TYPE ST_HW_InOutputsSTI_EtherCAT_Conveyor :
(**************************************************************************************
 * 	Application		:	BoxControl Framework
 *	Revision		:	$Revision: 355211 $
 *	Revision date	:	$Date: 2015-09-22 11:14:21 +0200 (Tue, 22 Sep 2015) $
 *	Last changed by	:	$Author: b7bolm $
 *	URL				:	$URL: http://almscdc.swisslog.com/repo/SWPD/Development/BoxControlFramework/20_Release/trunk/01_Software/BoxControlFramework/BoxControlFramework/JumpStart/11_Library/10_Application/11_Communication/12_MFCS/11_SIS/10_Base/FB_SIS_BaseDriver.TcPOU $
 *
 *	Purpose			:	Data for conveyor Subsystem interface over EtherCAT
 *
 * ------------------------------------------------------------------------------------
 *	Copyright Swisslog [IP AG], Switzerland. All rights reserved.
 * 
 * ------------------------------------------------------------------------------------
 *	
 * 	Revision History: 
 *
 * 	VERSION			DATE			INITIALS			DESCRIPTION
 *	0.1				01.01.2001		swl					Example
 *
 **************************************************************************************)
STRUCT
	Watchdog			: BOOL; // Communication supervision 
	FastSpeedActive		: BOOL; // Fast Speed Active
	TransportActive		: BOOL; // Transport Active
	Reserve1			: BOOL; // Reserve bit 
	Reserve2			: BOOL; // Reserve bit 
	Reserve3			: BOOL; // Reserve bit 
	Reserve4			: BOOL; // Reserve bit 
	Reserve5			: BOOL; // Reserve bit 
	
	TakeOverState 		: INT; // Takeover state
	HandOverState 		: INT; // Handover state 
	
	TU_ID				: STRING(Conveyor.TU_ID_STRINGLENGTH);
	Destination			: STRING(Conveyor.POSITION_STRINGLENGTH);
	AssignmentID		: UDINT;
	ExternalDeviceInOP	: BOOL; // External device in OP state
	State				: UINT;	// Ethercat State of the EL6695
END_STRUCT
END_TYPE

(* stored: Version 1.1.0.1, ProductVersion 3.1.4022.12
   DUT ST_HW_InOutputsSTI_EtherCAT_Conveyor: Id {c8780476-d44b-4943-921f-7ee0147594b1} *)
